// TwinCAT 3 PLC project Test_1
// ProgramVersion: 3.1.4024.0
// libraries:
//   Tc2_EtherCAT, * (Beckhoff Automation GmbH)
//   Tc2_Math, * (Beckhoff Automation GmbH)
//   Tc2_Standard, * (Beckhoff Automation GmbH)
//   Tc2_System, * (Beckhoff Automation GmbH)
//   Tc3_EventLogger, * (Beckhoff Automation GmbH)
//   Tc3_Module, * (Beckhoff Automation GmbH)
// project tree:
//   / PlcTask.TcTTO
//   POUs/ EventLogger_Alarms.TcPOU, EventLoggerManager.TcPOU, MAIN.TcPOU
// real-time tasks:
//   TASK PlcTask: cycle T#2ms, priority 4, ADS port 350

CONFIGURATION Test_1
    RESOURCE PLC ON TwinCAT3
        TASK PlcTask(INTERVAL := T#2ms, PRIORITY := 4);
        PROGRAM MAIN WITH PlcTask : MAIN;
    END_RESOURCE
END_CONFIGURATION

// ---- POUs/MAIN.TcPOU
PROGRAM MAIN
VAR

	SysRun					: BYTE;
	
END_VAR

SysRun := SysRun + 1;

EventLoggerManager();

RETURN;

END_PROGRAM

// ---- POUs/EventLoggerManager.TcPOU
PROGRAM EventLoggerManager
VAR
	Alarms						: EventLogger_Alarms;
	NumberOfAlarms				: INT;
	IsRunningToggle				: BOOL;
	AreAlarmsRaised				: ARRAY [1..2] OF BOOL;
	AlarmConfirmationStates		: ARRAY [1..2] OF TcEventConfirmationState;
	AlarmId						: UDINT := 1; // 1 = Main Door, 2 = Side Door, simple examples not linked to IO
	
	State						: INT;
	i							: INT;
	Result						: HRESULT;
END_VAR


// Manages the 'EventLogger_Alarms' object

// Change 'Id' to pick the alarm that will be interacted with (based on the ID of the Event Classes event, currently 1 or 2)
// Change 'State' to modify the alarms current state

Alarms.CyclicUpdate();

IsRunningToggle 			:= Alarms.Get_IsRunningToggle();
NumberOfAlarms 				:= Alarms.Get_AlarmCount();
AreAlarmsRaised 			:= Alarms.Get_AreAlarmsRaised();
AlarmConfirmationStates 	:= Alarms.Get_ConfirmationStates();

CASE State OF
	
	0:
		;
		
	1: // Raise
		Result := Alarms.TriggerAlarm(AlarmId := AlarmId);
		State := 0;
		
	2: // Confirm
		Result := Alarms.ConfirmAlarm(AlarmId := AlarmId);
		State := 0;
		
	3: // Clear
		Result := Alarms.ClearAlarm(AlarmId := AlarmId, ResetConfirmationState := TRUE);
		State := 0;

END_CASE

RETURN;

END_PROGRAM

// ---- POUs/EventLogger_Alarms.TcPOU
// Manages an Event Class, creates an alarm for each Event in the class which can be controlled

// Uses Event Class pre-made in the 'Type System': called 'PersonalEventLogger'
// Uses Events pre-made in the 'Event Class'
// Number of events must be manually defined in '_EventCount'
// Severity of events must be manually defined in '_EventSeverity'

{attribute 'no_explicit_call' := 'Do not call this block directly, use the METHODS this block has'}
FUNCTION_BLOCK EventLogger_Alarms
VAR
	
	_IsRunningToggle		: BOOL;
	_i						: INT;
	
	_Alarm					: ARRAY [1.._EventCount] OF FB_TcAlarm;
	_IsConfirmationNeeded	: ARRAY [1.._EventCount] OF BOOL;
	_Event					: ARRAY [1.._EventCount] OF TcEventEntry;
	_EventSeverity			: ARRAY [1.._EventCount] OF TcEventSeverity := 
								// Manually enter the severity of each alarm here:
								[TcEventSeverity.Error, 
								 TcEventSeverity.Warning];
	
END_VAR
VAR CONSTANT
	
	_EventCount				: INT := 2;

END_VAR

METHOD ClearAlarm : HRESULT
VAR_INPUT
	AlarmId						: UDINT;
	ResetConfirmationState		: BOOL;
END_VAR

// Clears an alarm 

ClearAlarm := _Alarm[AlarmId].Clear(nTimeStamp := 0, bResetConfirmation := ResetConfirmationState);
RETURN;
END_METHOD

METHOD ConfirmAlarm : HRESULT
VAR_INPUT
	AlarmId		: UDINT;
END_VAR

// Acknowledges an alarm 
// This does not clear the alarm
// This does change the alarms state internally

ConfirmAlarm := _Alarm[AlarmId].Confirm(nTimeStamp := 0);
RETURN;
END_METHOD

METHOD CyclicUpdate : BOOL

_IsRunningToggle := NOT(_IsRunningToggle);
RETURN;
END_METHOD

{attribute 'no_explicit_call' := 'You do not need to use this METHOD'}
METHOD FB_init : BOOL 
VAR_INPUT
	bInitRetains : BOOL; // if TRUE, the retain variables are initialized (warm start / cold start)
	bInCopyCode : BOOL;  // if TRUE, the instance afterwards gets moved into the copy code (online change)
END_VAR

// Initialise the event parameters and then the alarms that are tied to the events

FOR _i := 1 TO _EventCount BY 1 DO
	
	// All alarms need confirmation
	_IsConfirmationNeeded[_i] := TRUE;
	
END_FOR

FOR _i := 1 TO _EventCount BY 1 DO
	
	// Defining event settings / parameters
	_Event[_i].uuidEventClass 		:= TC_EVENT_CLASSES.PersonalEventLogger;
	_Event[_i].nEventId 			:= INT_TO_UDINT(_i);
	_Event[_i].eSeverity			:= _EventSeverity[_i];
	
	// Important to set both the Events eFlag and the Alarms bWithConfirmation to the same bool value
	_Event[_i].eFlags 				:= BOOL_TO_BYTE(_IsConfirmationNeeded[_i]);
	
END_FOR

FOR _i := 1 TO _EventCount BY 1 DO

	_Alarm[_i].CreateEx
	(
		stEventEntry := _Event[_i],
		ipSourceInfo := 0,
		
		// Important to set both the Events eFlag and the Alarms bWithConfirmation to the same bool value
		bWithConfirmation := _IsConfirmationNeeded[_i]
	);	

END_FOR

RETURN;
END_METHOD

METHOD Get_AlarmCount : INT // Returns the number of alarms that exist

Get_AlarmCount := _EventCount;
RETURN;
END_METHOD

METHOD Get_AreAlarmsRaised : ARRAY [1.._EventCount] OF BOOL // Returns an array of BOOLS to represent if an alarm is raised

FOR _i := 1 TO _EventCount DO
    Get_AreAlarmsRaised[_i] := _Alarm[_i].bRaised;
END_FOR
RETURN;
END_METHOD

METHOD Get_ConfirmationStates : ARRAY [1.._EventCount] OF TcEventConfirmationState // Returns an array of confirmation states of alarms

FOR _i := 1 TO _EventCount DO
    Get_ConfirmationStates[_i] := _Alarm[_i].eConfirmationState;
END_FOR
RETURN;
END_METHOD

METHOD Get_IsRunningToggle : BOOL // Returns a BOOL that toggles states when the object's cyclic update is running
VAR_INPUT
END_VAR

Get_IsRunningToggle := _IsRunningToggle;
RETURN;
END_METHOD

METHOD TriggerAlarm : HRESULT
VAR_INPUT
	AlarmId		: UDINT;
END_VAR

// Triggers an alarm

TriggerAlarm := _Alarm[AlarmId].Raise(nTimeStamp := 0);
RETURN;
END_METHOD

END_FUNCTION_BLOCK
